// TIA Portal V18 export
DATA_BLOCK "level"   // DB72
{ S7_Optimized_Access := 'TRUE' }
VERSION : 0.1
// stored: AutoNumber true, DBAccessibleFromOPCUA true, IsOnlyStoredInLoadMemory false, IsRetainMemResEnabled false, IsWriteProtectedInAS false, MemoryReserve 100
   VAR RETAIN
      "A" : Struct
         "Low level" : Real := 20.0;
         "high level" : Real := 90.0;
         "level empty" : Real := 10.0;
      END_STRUCT;
      "B" : Struct
         "Low level" : Real := 20.0;
         "high level" : Real := 90.0;
         "level empty" : Real := 10.0;
      END_STRUCT;
      "present A1" : Real;
      "present A2" : Real;
      "present B1" : Real;
      "present B2" : Real;
   END_VAR
   VAR
      "Low level occured A1" : Bool;
      "Low level occured A2" : Bool;
      "High Level A" : Bool;
      "High Level B" : Bool;
      "Level Empty A2" : Bool;
      "Level Empty A1" : Bool;
      "Low level occured B1" : Bool;
      "Low level occured B2" : Bool;
      "Level Empty B1" : Bool;
      "Level Empty B2" : Bool;
      "Active vessel A" : Int;
      "Active vessel B" : Int;
      "scale A1" : Struct
         NormX : Real;
         scalx : Real;
      END_STRUCT;
      "scale B1" : Struct
         NormX : Real;
         scalx : Real;
      END_STRUCT;
      "Low level occured A" : Bool;
      "Low level occured B" : Bool;
      "Level Empty A" : Bool;
      "Level Empty B" : Bool;
      "Catridge low level A" : Bool;
      "Catridge low level B" : Bool;
      "Catridge level empty A" : Bool;
      "Catridge level empty B" : Bool;
      "Drum Level Low A1" : Bool;
      "Drum Level Low A2" : Bool;
      "Drum Level Empty A1" : Bool;
      "Drum Level Empty A2" : Bool;
      "Drum Level Low B1" : Bool;
      "Drum Level Low B2" : Bool;
      "Drum Level Empty B1" : Bool;
      "Drum Level Empty B2" : Bool;
   END_VAR
BEGIN
END_DATA_BLOCK
